FUNCTION F_ROUND_REAL_GLOBAL : ARRAY[1..6] OF REAL
VAR_INPUT
  iDecimalPlaces 	: INT;
END_VAR
VAR
  rOutput 			: ARRAY[1..6] OF REAL;
  Value				: ARRAY[1..6] OF DINT;
  X					: int;
END_VAR

FOR X := 1 TO 6 BY 1 DO
	rOutput[X] := LREAL_TO_REAL(GVL.rRawValue[X] * EXPT(10,iDecimalPlaces));
	Value[X] := REAL_TO_DINT(rOutput[X]);
	rOutput[X] := LREAL_to_real(Value[X] / EXPT(10,iDecimalPlaces));
END_FOR

F_ROUND_REAL_GLOBAL := rOutput;

END_FUNCTION

(* stored: Version 1.1.0.1, ProductVersion 3.1.4024.12
   POU F_ROUND_REAL_GLOBAL: Id {967fe789-c289-4fa6-aeef-63816f5b0f8e}, SpecialFunc None *)
